Staubli VAL3: SETVIEW.pgx

public program setView(bool x_bLarge)
begin
  //-----------------------------------------------------------------------
  //Header begin
  //Description of program
  //  Allows enlarging the width of the list menu. After called this
  //  program, you will regenerate your interface.
  //
  //Input parameters
  //  bool x_bLarge :
  //    role : For enlarge the width of the list menu.
  //    posssible value : true  => enlarge the width of the list menu
  //                      false => normal width (width defines with setSizeList)
  //
  //Example
  //  call x_bLarge(true)
  //
  //History
  //  Creation : 28-04-08 - f.Rob
  //Header end
  //-----------------------------------------------------------------------
  //Save the TopX position in an other element
  //Put TopX width on the maximum (38) for enlarge the list menu
  if x_bLarge
    nTopX[1]=nTopX
    nTopX=0
    nBottomX[1]=nBottomX
    nBottomX=38
  else
    //Restore the TopX position saved
    nTopX=nTopX[1]
    nBottomX=nBottomX[1]
  endIf
  bUseRefresh=true
end
